// TIA Portal V17 export
// export: Created 2025-03-05T08:02:13.0792508Z, ExportSetting WithDefaults, DisplayName Totally Integrated Automation Portal, DisplayVersion V17 Update 8, DisplayName TIA Portal Openness, DisplayVersion V17 Update 8, DisplayName TIA Portal Version Control Interface, DisplayVersion V17, DisplayName SINAMICS Startdrive Advanced, DisplayVersion V17 SP2, DisplayName SINAMICS Startdrive G110M, G120, G120C, G120D, G120P, G115D, DisplayVersion V17 SP2, DisplayName SINAMICS Startdrive G130, G150, S120, S150, SINAMICS MV, S210, DisplayVersion V17 SP2, DisplayName STEP 7 Professional, DisplayVersion V17 Update 8, DisplayName SINUMERIK ONE STEP 7 Toolbox, DisplayVersion V17 Update 12, DisplayName SINUMERIK 840D sl STEP 7 Toolbox, DisplayVersion V17 Update 12, DisplayName STEP 7 Safety, DisplayVersion V17 Update 6, DisplayName WinCC Advanced, DisplayVersion V17 Update 8
TYPE "AXIS_SAFETY_OUT"
// stored: IsFailsafeCompliant true
   STRUCT
      Deselect_STO : Bool;   // DESELECT SAFE TORQUE OFF
      Deselect_SS1 : Bool;   // DESELECT SAFE STOP 1
      Deselect_SS2 : Bool;   // DESELECT SAFE STOP 2
      Deselect_SOS : Bool;   // DESELECT SAFE OPERATING STOP
      Deselect_SLS : Bool;   // DESELECT SAFE LIMITED SPEED
      Reserved_Out_1 : Bool;
      Deselect_SLP : Bool;   // DESELECT SAFETY LOGIC PROGRAMME
      Ack_Inc_Event : Bool;   // ACKNOWLEDGE INTERNAL EVENT ACTIVE
      Reserved_Out_2 : Bool;
      Select_SLS_bit_0 : Bool;   // SELECT SAFE LIMITED SPEED BIT 0
      Select_SLS_bit_1 : Bool;   // SELECT SAFE LIMITED SPEED BIT 1
      Reserved_Out_3 : Bool;
      Deselect_SDI_Pos : Bool;   // DESELECT SAFE DIRECTION POSITIVE
      Deselect_SDI_Neg : Bool;   // DESELECT SAFE DIRECTION NEGATIVE
      Reserved_Out_4 : Bool;
      Reserved_Out_5 : Bool;
      Reserved_Out_6 : Bool;
      Reserved_Out_7 : Bool;
      Reserved_Out_8 : Bool;
      Select_SPL_range : Bool;   // SELECT SAFETY LOGIC PROGRAMME RANGE
      Reserved_Out_9 : Bool;
      Reserved_Out_10 : Bool;
      Reserved_Out_11 : Bool;
      Des_Safe_Cam : Bool;   // DESELECT SAFETY CAMS
      Select_Gear_bit_0 : Bool;   // SELECT GEAR BIT 0
      Select_Gear_bit_1 : Bool;   // SELECT GEAR BIT 1
      Select_Gear_bit_2 : Bool;   // SELECT GEAR BIT 2
      Deselect_Gear_Sw : Bool;   // DESELECT GEAR SW
      Deselect_SS2E : Bool;   // DESELECT SAFE STOP 2 EXTENDED
      Deselect_SS2ESR : Bool;   // DESELECT SAFE STOP 2 EXTENDED ESR
      Reserved_Out_14 : Bool;   // DESELECT
      Reserved_Out_15 : Bool;   // DESELECT
      SLS1_Limit : Word;   // SAFELY LIMITED SPEED 1 LIMIT
   END_STRUCT;
END_TYPE
